// TIA Portal V19 export
TYPE "CTRL_CVLV"
   STRUCT
      status : Bool;
      sim : "UDT_SIM_VLV";
   END_STRUCT;
END_TYPE
